{attribute 'pack_mode' := '1'}
TYPE ST_MoveVehicleStatusDataIn :
STRUCT
	iCommandID					: UINT;													// The command ID for this command

END_STRUCT
END_TYPE

(* stored: Version 1.1.0.1, ProductVersion 3.1.4024.5
   DUT ST_MoveVehicleStatusDataIn: Id {3803fd8b-1bb8-4cde-93bc-9eebac4f5602} *)
